{attribute addProperty BoxType "EK1122-0000-0018"}
{attribute addProperty Id "Beckhoff_AX8yxxsub_EK1100EK1100_179A0949162A_0061_AMP8000_0000_0103AMP8000_2B90571139449.25A_0061_AMP8000_0030_0103AMP8000_5E0E86F855669.5"}
{attribute addProperty CRC "1572356787"}
{attribute addProperty SizeInBites "966"}
{attribute addProperty SizeInBytes "120.75"}
TYPE Beckhoff_AX8yxxEK1122_5DB842B3 EXTENDS EK1122_179A0949 :
STRUCT
	{attribute addProperty Name "Beckhoff_AX8yxxsub_EK1100"}
	Beckhoff_AX8yxxsub_EK1100 : EK1100_179A0949;
	{attribute addProperty Name "A_0061_AMP8000_0000_0103"}
	A_0061_AMP8000_0000_0103 : AMP8000_2B905711;
	{attribute addProperty Name "A_0061_AMP8000_0030_0103"}
	A_0061_AMP8000_0030_0103 : AMP8000_5E0E86F8;
END_STRUCT
END_TYPE

(* stored: Version 1.2.0.0, ProductVersion 3.1.4024.9
   DUT Beckhoff_AX8yxxEK1122_5DB842B3: Id {9d0f0586-4818-4775-8123-b6fbf18b72b4} *)
